// TIA Portal project "1200客户机" (V12)

(* hardware
DEVICE "S7-1200 station_1"  SIMATIC 1200-Station
   slot 0: "S7-1200 机架"  Rack  V1.0
   slot 1: "PLC_1"  CPU 1214C AC/DC/Rly  6ES7 214-1BE30-0XB0  V2.2
*)

// ===== PLC "PLC_1"  CPU 1214C AC/DC/Rly =====

VAR_GLOBAL   // PLC tag table "默认变量表"
   "Tag_1" AT %M8.1 : Bool;
   "Tag_2" AT %M10.0 : Bool;
   "Tag_3" AT %M0.1 : Bool;
   "Tag_4" AT %M0.2 : Bool;
   "Tag_5" AT %MW2 : Word;
   "Tag_6" AT %M10.1 : Bool;
   "Tag_7" AT %M10.2 : Bool;
   "Tag_8" AT %MW12 : Word;
   "Clock_Byte" AT %MB8 : Byte;
   "Clock_10Hz" AT %M8.0 : Bool;
   "Clock_2Hz" AT %M8.3 : Bool;
   "Clock_1.25Hz" AT %M8.4 : Bool;
   "Clock_1Hz" AT %M8.5 : Bool;
   "Clock_0.625Hz" AT %M8.6 : Bool;
   "Clock_0.5Hz" AT %M8.7 : Bool;
   "Tag_9" AT %MW204 : UInt;
   "Tag_10" AT %MW4 : UInt;
END_VAR

DATA_BLOCK "Data_block_1"   // DB1
{ S7_Optimized_Access := 'FALSE' }
VERSION : 0.1
   VAR
      ARAY : Array [0 .. 99] of Int;
   END_VAR
BEGIN
END_DATA_BLOCK

DATA_BLOCK "Data_block_2"   // DB2
{ S7_Optimized_Access := 'FALSE' }
VERSION : 0.1
   VAR
      ARAY : Array [0 .. 99] of  Int;
   END_VAR
BEGIN
END_DATA_BLOCK

ORGANIZATION_BLOCK "Main"   // OB1, LAD, ProgramCycle
TITLE = "Main Program Sweep (Cycle)"
{ S7_Optimized_Access := 'FALSE' }
VERSION : 0.1
BEGIN

REGION Network 1
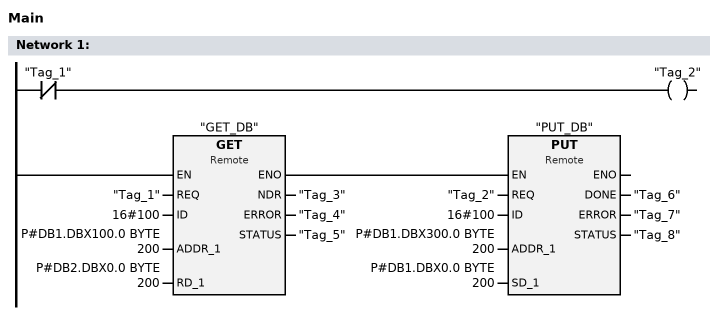
   // ENO of a box is taken as its EN; it also drops when the box reports an error
   "Tag_2" := NOT "Tag_1";
   "GET_DB"(REQ := "Tag_1",   // GET
            ID := 16#100,
            ADDR_1 := P#DB1.DBX100.0 BYTE 200,
            RD_1 := P#DB2.DBX0.0 BYTE 200,
            NDR => "Tag_3",
            ERROR => "Tag_4",
            STATUS => "Tag_5");
   "PUT_DB"(REQ := "Tag_2",   // PUT
            ID := 16#100,
            ADDR_1 := P#DB1.DBX300.0 BYTE 200,
            SD_1 := P#DB1.DBX0.0 BYTE 200,
            DONE => "Tag_6",
            ERROR => "Tag_7",
            STATUS => "Tag_8");
END_REGION
END_ORGANIZATION_BLOCK

ORGANIZATION_BLOCK "Cyclic interrupt"   // OB30, LAD, CyclicInterrupt
{ S7_Optimized_Access := 'FALSE' }
VERSION : 0.1
BEGIN

REGION Network 1
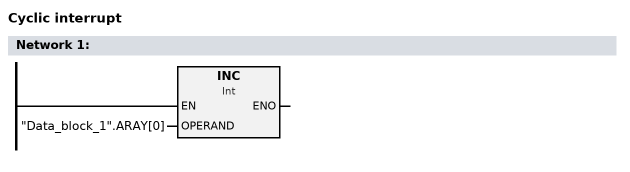
   RUNG wire#powerrail
      { S7_Templates := "DestType := Int"; S7_GenerateENO := "TRUE" } Inc( "Data_block_1".ARAY[0] )
   END_RUNG
   // the same network as SCL:
   "Data_block_1".ARAY[0] := "Data_block_1".ARAY[0] + 1;
END_REGION

REGION Network 2: [
END_REGION
END_ORGANIZATION_BLOCK

ORGANIZATION_BLOCK "Startup"   // OB100, LAD, Startup
TITLE = "Complete Restart"
{ S7_Optimized_Access := 'FALSE' }
VERSION : 0.1
   VAR_INPUT
      LostRetentive : Bool;   // True if retentive data are lost
      LostRTC : Bool;   // True if date and time are lost
   END_VAR
BEGIN

REGION Network 1
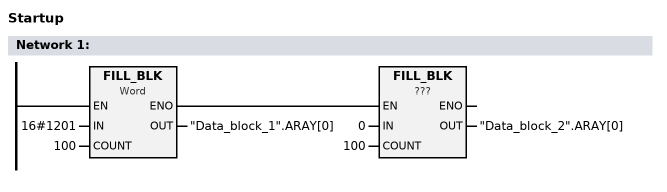
   RUNG wire#powerrail
      { S7_Templates := "CountType := Word"; S7_GenerateENO := "TRUE" } FillBlockI(in := 16#1201, count := 100, out => "Data_block_1".ARAY[0])
      { S7_Templates := "CountType := ???"; S7_GenerateENO := "TRUE" } FillBlockI(in := 0, count := 100, out => "Data_block_2".ARAY[0])
   END_RUNG
   // the same network as SCL:
   // ENO of a box is taken as its EN; it also drops when the box reports an error
   FILL_BLK(IN := 16#1201, COUNT := 100, OUT => "Data_block_1".ARAY[0]);
   FILL_BLK(IN := 0, COUNT := 100, OUT => "Data_block_2".ARAY[0]);
END_REGION
END_ORGANIZATION_BLOCK